{attribute 'GeneratedUsingTerminal: EL3443-0000-0016'}
{attribute addProperty BoxType "EL3443-0000-0016"}
{attribute addProperty Id "L1_L2_VoltageAT %I*REAL4L2_L3_VoltageAT %I*REAL4L3_L1_VoltageAT %I*REAL4"}
{attribute addProperty CRC "679556377"}
{attribute addProperty Size "12"}
TYPE Total_L_L_Voltage_28813519 EXTENDS InputBase_8311D824 :
STRUCT
	{attribute addProperty Name "L1_L2_Voltage"}
	L1_L2_Voltage AT %I* : REAL;
	{attribute addProperty Name "L2_L3_Voltage"}
	L2_L3_Voltage AT %I* : REAL;
	{attribute addProperty Name "L3_L1_Voltage"}
	L3_L1_Voltage AT %I* : REAL;
END_STRUCT
END_TYPE

(* stored: Version 1.2.0.0, ProductVersion 3.1.4024.11
   DUT Total_L_L_Voltage_28813519: Id {c3982ee9-b5b7-45bf-b63a-ad12ef1617d9} *)
